PROGRAM Postman_filter
VAR

    sJsonResponse  : STRING(255);
    sCleanedJson   : STRING(255);
    sReplaceWith   : STRING(255);
    iPos           : INT;
    sKeyToFind     : STRING(255);
    iStartPos      : INT;
    iEndPos        : INT;
    sTempString    : STRING(255);
    sContainerCode : STRING(255);
	iPos2		   : INT := 0;
END_VAR


// Example JSON with $N
sJsonResponse := IO.sMES_binID;
sCleanedJson := sJsonResponse;
sReplaceWith := ' ';

// Replace all occurrences of $N with a space
iPos := FIND(sCleanedJson, '$N');
WHILE iPos > 0 DO
    // REPLACE signature: REPLACE(STR1, STR2, L, P)
    // L = 2 (because '$N' has length 2)
    // P = iPos (position from FIND)
    sCleanedJson := REPLACE(sCleanedJson, sReplaceWith, 2, iPos);
    iPos := FIND(sCleanedJson, '$N');
END_WHILE;

// Now sCleanedJson should have no $N. It should look like a clean JSON string.

// Next, find the "ContainerCode"
sKeyToFind := '\"ContainerCode\":';
iPos := FIND(sCleanedJson, sKeyToFind);
IF iPos > 0 THEN
    iStartPos := iPos + LEN(sKeyToFind); // Move past "ContainerCode":
    iStartPos := iStartPos + 2;          // Skip the opening quote for the value

    sTempString := MID(sCleanedJson, LEN(sCleanedJson) - iStartPos + 1, iStartPos );

    iEndPos := FIND(sTempString, '"');
    IF iEndPos > 0 THEN
        sContainerCode := MID(sTempString, (iEndPos - 1), 1);
    ELSE
        sContainerCode := '';
    END_IF
ELSE
    sContainerCode := '';
END_IF;

IO.sReceiving_binID := sContainerCode;


iPos2 := FIND(IO.sReceiving_binID, '\');
WHILE iPos2 > 0 DO
    IO.sReceiving_binID := REPLACE(IO.sReceiving_binID, '', 1, iPos2); // Replace one '\' char with empty string
    iPos2 := FIND(IO.sReceiving_binID, '\');
END_WHILE;

END_PROGRAM

(* stored: Version 1.1.0.1, ProductVersion 3.1.4024.12
   POU Postman_filter: Id {fa700dfb-6b48-49e8-a364-c9f0219799d7}, SpecialFunc None *)
